ABB RAPID module: Module1.mod

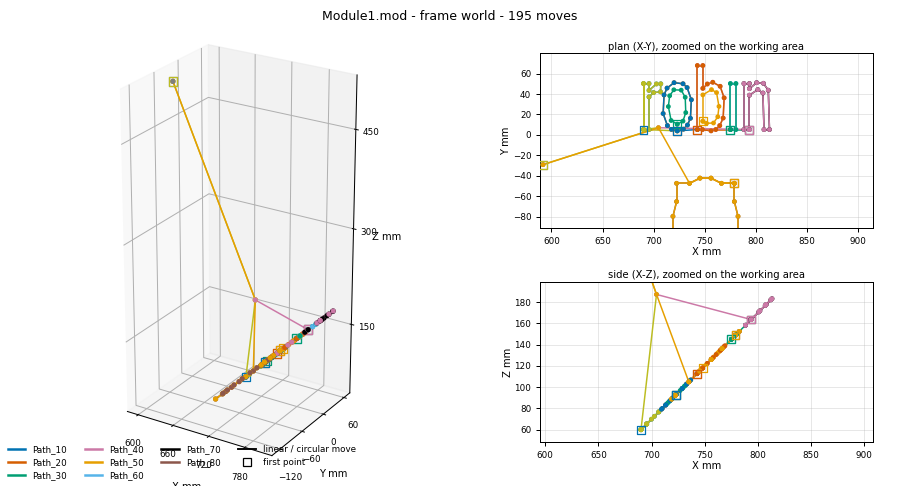
[picture p0: tool path of Module1.mod in frame world, 195 of 195 moves have a stored position in this frame; points joined in program order, loops and branches not executed]
MODULE Module1
        CONST robtarget Target_10:=[[-207.881930308,149.087746467,0.000160807],[0.518535839,0.510701659,-0.288134644,0.622320517],[0,0,1,1],[9E+09,9E+09,9E+09,9E+09,9E+09,9E+09]];
    CONST robtarget Target_20:=[[-247.65501993,195.765129088,0.000181206],[0.450409444,-0.243963603,-0.202089765,-0.83472919],[0,0,0,0],[9E+09,9E+09,9E+09,9E+09,9E+09,9E+09]];
    CONST robtarget Target_30:=[[-247.65501993,188.180039946,0.000181208],[0.450409444,-0.243963603,-0.202089765,-0.83472919],[0,0,0,0],[9E+09,9E+09,9E+09,9E+09,9E+09,9E+09]];
    CONST robtarget Target_40:=[[-240.945133383,188.180039946,0.000181208],[0.450409444,-0.243963603,-0.202089765,-0.83472919],[0,0,0,0],[9E+09,9E+09,9E+09,9E+09,9E+09,9E+09]];
    CONST robtarget Target_50:=[[-247.278196592,177.914642864,0.000181211],[0.450409444,-0.243963603,-0.202089765,-0.83472919],[0,0,0,0],[9E+09,9E+09,9E+09,9E+09,9E+09,9E+09]];
    CONST robtarget Target_60:=[[-247.411908099,171.89154724,0.000181212],[0.450409444,-0.243963603,-0.202089765,-0.83472919],[0,0,0,0],[9E+09,9E+09,9E+09,9E+09,9E+09,9E+09]];
    CONST robtarget Target_70:=[[-239.53508476,172.28052617,0.000181212],[0.450409444,-0.243963603,-0.202089765,-0.83472919],[0,0,0,0],[9E+09,9E+09,9E+09,9E+09,9E+09,9E+09]];
    CONST robtarget Target_80:=[[-238.811255907,181.791619828,0.00018121],[0.450409444,-0.243963603,-0.202089765,-0.83472919],[0,0,0,0],[9E+09,9E+09,9E+09,9E+09,9E+09,9E+09]];
    CONST robtarget Target_90:=[[-234.575603399,188.180039946,0.000181208],[0.450409444,-0.243963603,-0.202089765,-0.83472919],[0,0,0,0],[9E+09,9E+09,9E+09,9E+09,9E+09,9E+09]];
    CONST robtarget Target_100:=[[-202.630708747,188.180039946,0.000181208],[0.450409444,-0.243963603,-0.202089765,-0.83472919],[0,0,0,0],[9E+09,9E+09,9E+09,9E+09,9E+09,9E+09]];
    CONST robtarget Target_110:=[[-202.630708747,195.765129088,0.000181206],[0.450409444,-0.243963603,-0.202089765,-0.83472919],[0,0,0,0],[9E+09,9E+09,9E+09,9E+09,9E+09,9E+09]];
    CONST robtarget Target_120:=[[-201.366527224,149.087657451,0.000181219],[0.450409444,-0.243963603,-0.202089765,-0.83472919],[0,0,0,0],[9E+09,9E+09,9E+09,9E+09,9E+09,9E+09]];
    CONST robtarget Target_130:=[[-203.021765343,140.621098181,0.000181221],[0.450409444,-0.243963603,-0.202089765,-0.83472919],[0,0,0,0],[9E+09,9E+09,9E+09,9E+09,9E+09,9E+09]];
    CONST robtarget Target_140:=[[-207.051498291,134.946923266,0.000181223],[0.450409444,-0.243963603,-0.202089765,-0.83472919],[0,0,0,0],[9E+09,9E+09,9E+09,9E+09,9E+09,9E+09]];
    CONST robtarget Target_150:=[[-213.680713864,130.849034031,0.000181224],[0.450409444,-0.243963603,-0.202089765,-0.83472919],[0,0,0,0],[9E+09,9E+09,9E+09,9E+09,9E+09,9E+09]];
    CONST robtarget Target_160:=[[-231.788173899,129.551975923,0.000181224],[0.450409444,-0.243963603,-0.202089765,-0.83472919],[0,0,0,0],[9E+09,9E+09,9E+09,9E+09,9E+09,9E+09]];
    CONST robtarget Target_170:=[[-243.683087922,135.407213167,0.000181223],[0.450409444,-0.243963603,-0.202089765,-0.83472919],[0,0,0,0],[9E+09,9E+09,9E+09,9E+09,9E+09,9E+09]];
    CONST robtarget Target_180:=[[-247.461911379,141.100681452,0.000181221],[0.450409444,-0.243963603,-0.202089765,-0.83472919],[0,0,0,0],[9E+09,9E+09,9E+09,9E+09,9E+09,9E+09]];
    CONST robtarget Target_190:=[[-248.515109012,153.46115467,0.000181218],[0.450409444,-0.243963603,-0.202089765,-0.83472919],[0,0,0,0],[9E+09,9E+09,9E+09,9E+09,9E+09,9E+09]];
    CONST robtarget Target_200:=[[-243.220985991,163.168323786,0.000181215],[0.450409444,-0.243963603,-0.202089765,-0.83472919],[0,0,0,0],[9E+09,9E+09,9E+09,9E+09,9E+09,9E+09]];
    CONST robtarget Target_210:=[[-236.515653903,167.360178067,0.000181214],[0.450409444,-0.243963603,-0.202089765,-0.83472919],[0,0,0,0],[9E+09,9E+09,9E+09,9E+09,9E+09,9E+09]];
    CONST robtarget Target_220:=[[-218.290970645,168.613376793,0.000181213],[0.450409444,-0.243963603,-0.202089765,-0.83472919],[0,0,0,0],[9E+09,9E+09,9E+09,9E+09,9E+09,9E+09]];
    CONST robtarget Target_230:=[[-206.527619769,162.711873191,0.000181215],[0.450409444,-0.243963603,-0.202089765,-0.83472919],[0,0,0,0],[9E+09,9E+09,9E+09,9E+09,9E+09,9E+09]];
    CONST robtarget Target_240:=[[-202.813142148,157.107360988,0.000181217],[0.450409444,-0.243963603,-0.202089765,-0.83472919],[0,0,0,0],[9E+09,9E+09,9E+09,9E+09,9E+09,9E+09]];
    CONST robtarget Target_250:=[[-201.366527224,149.087657451,0.000181219],[0.450409444,-0.243963603,-0.202089765,-0.83472919],[0,0,0,0],[9E+09,9E+09,9E+09,9E+09,9E+09,9E+09]];
    CONST robtarget Target_450:=[[-207.881924306,149.087657451,0.000181219],[0.450409444,-0.243963603,-0.202089765,-0.83472919],[0,0,0,0],[9E+09,9E+09,9E+09,9E+09,9E+09,9E+09]];
    CONST robtarget Target_460:=[[-210.90124058,141.155060399,0.000181221],[0.450409444,-0.243963603,-0.202089765,-0.83472919],[0,0,0,0],[9E+09,9E+09,9E+09,9E+09,9E+09,9E+09]];
    CONST robtarget Target_470:=[[-219.222672222,137.293167892,0.000181222],[0.450409444,-0.243963603,-0.202089765,-0.83472919],[0,0,0,0],[9E+09,9E+09,9E+09,9E+09,9E+09,9E+09]];
    CONST robtarget Target_480:=[[-234.22183773,138.044318657,0.000181223],[0.450409444,-0.243963603,-0.202089765,-0.83472919],[0,0,0,0],[9E+09,9E+09,9E+09,9E+09,9E+09,9E+09]];
    CONST robtarget Target_490:=[[-241.204901386,143.601825103,0.00018122],[0.450409444,-0.243963603,-0.202089765,-0.83472919],[0,0,0,0],[9E+09,9E+09,9E+09,9E+09,9E+09,9E+09]];
    CONST robtarget Target_500:=[[-241.55017581,153.821736994,0.000181218],[0.450409444,-0.243963603,-0.202089765,-0.83472919],[0,0,0,0],[9E+09,9E+09,9E+09,9E+09,9E+09,9E+09]];
    CONST robtarget Target_510:=[[-235.724815439,159.591250126,0.000181216],[0.450409444,-0.243963603,-0.202089765,-0.83472919],[0,0,0,0],[9E+09,9E+09,9E+09,9E+09,9E+09,9E+09]];
    CONST robtarget Target_520:=[[-225.142864339,161.389116121,0.000181215],[0.450409444,-0.243963603,-0.202089765,-0.83472919],[0,0,0,0],[9E+09,9E+09,9E+09,9E+09,9E+09,9E+09]];
    CONST robtarget Target_530:=[[-211.506651645,157.581568731,0.000181217],[0.450409444,-0.243963603,-0.202089765,-0.83472919],[0,0,0,0],[9E+09,9E+09,9E+09,9E+09,9E+09,9E+09]];
    CONST robtarget Target_540:=[[-207.881924306,149.087657451,0.000181219],[0.450409444,-0.243963603,-0.202089765,-0.83472919],[0,0,0,0],[9E+09,9E+09,9E+09,9E+09,9E+09,9E+09]];
    CONST robtarget Target_550:=[[-202.630708747,121.227041567,0.000181228],[0.450409444,-0.243963603,-0.202089765,-0.83472919],[0,0,0,0],[9E+09,9E+09,9E+09,9E+09,9E+09,9E+09]];
    CONST robtarget Target_560:=[[-202.630708747,114.128176089,0.000181229],[0.450409444,-0.243963603,-0.202089765,-0.83472919],[0,0,0,0],[9E+09,9E+09,9E+09,9E+09,9E+09,9E+09]];
    CONST robtarget Target_570:=[[-201.366527224,102.264318715,0.000181232],[0.450409444,-0.243963603,-0.202089765,-0.83472919],[0,0,0,0],[9E+09,9E+09,9E+09,9E+09,9E+09,9E+09]];
    CONST robtarget Target_580:=[[-202.647957508,95.740722444,0.000181234],[0.450409444,-0.243963603,-0.202089765,-0.83472919],[0,0,0,0],[9E+09,9E+09,9E+09,9E+09,9E+09,9E+09]];
    CONST robtarget Target_590:=[[-206.492248362,90.253373046,0.000181236],[0.450409444,-0.243963603,-0.202089765,-0.83472919],[0,0,0,0],[9E+09,9E+09,9E+09,9E+09,9E+09,9E+09]];
    CONST robtarget Target_600:=[[-213.89225132,85.531430921,0.000181237],[0.450409444,-0.243963603,-0.202089765,-0.83472919],[0,0,0,0],[9E+09,9E+09,9E+09,9E+09,9E+09,9E+09]];
    CONST robtarget Target_610:=[[-233.637220258,84.167137,0.000181237],[0.450409444,-0.243963603,-0.202089765,-0.83472919],[0,0,0,0],[9E+09,9E+09,9E+09,9E+09,9E+09,9E+09]];
    CONST robtarget Target_620:=[[-244.963719116,89.701429516,0.000181236],[0.450409444,-0.243963603,-0.202089765,-0.83472919],[0,0,0,0],[9E+09,9E+09,9E+09,9E+09,9E+09,9E+09]];
    CONST robtarget Target_630:=[[-248.919201454,99.881822767,0.000181233],[0.450409444,-0.243963603,-0.202089765,-0.83472919],[0,0,0,0],[9E+09,9E+09,9E+09,9E+09,9E+09,9E+09]];
    CONST robtarget Target_640:=[[-247.217418634,107.442600725,0.000181231],[0.450409444,-0.243963603,-0.202089765,-0.83472919],[0,0,0,0],[9E+09,9E+09,9E+09,9E+09,9E+09,9E+09]];
    CONST robtarget Target_650:=[[-242.9386504,113.641952426,0.000181229],[0.450409444,-0.243963603,-0.202089765,-0.83472919],[0,0,0,0],[9E+09,9E+09,9E+09,9E+09,9E+09,9E+09]];
    CONST robtarget Target_660:=[[-265.304938893,113.641952426,0.000181229],[0.450409444,-0.243963603,-0.202089765,-0.83472919],[0,0,0,0],[9E+09,9E+09,9E+09,9E+09,9E+09,9E+09]];
    CONST robtarget Target_670:=[[-265.304938893,121.227041567,0.000181228],[0.450409444,-0.243963603,-0.202089765,-0.83472919],[0,0,0,0],[9E+09,9E+09,9E+09,9E+09,9E+09,9E+09]];
    CONST robtarget Target_680:=[[-202.630708747,121.227041567,0.000181228],[0.450409444,-0.243963603,-0.202089765,-0.83472919],[0,0,0,0],[9E+09,9E+09,9E+09,9E+09,9E+09,9E+09]];
    CONST robtarget Target_760:=[[-210.750643917,113.641952426,0.000181229],[0.450409444,-0.243963603,-0.202089765,-0.83472919],[0,0,0,0],[9E+09,9E+09,9E+09,9E+09,9E+09,9E+09]];
    CONST robtarget Target_770:=[[-236.569120417,113.641952426,0.000181229],[0.450409444,-0.243963603,-0.202089765,-0.83472919],[0,0,0,0],[9E+09,9E+09,9E+09,9E+09,9E+09,9E+09]];
    CONST robtarget Target_780:=[[-241.723091243,101.68085032,0.000181232],[0.450409444,-0.243963603,-0.202089765,-0.83472919],[0,0,0,0],[9E+09,9E+09,9E+09,9E+09,9E+09,9E+09]];
    CONST robtarget Target_790:=[[-238.824332003,94.685562215,0.000181234],[0.450409444,-0.243963603,-0.202089765,-0.83472919],[0,0,0,0],[9E+09,9E+09,9E+09,9E+09,9E+09,9E+09]];
    CONST robtarget Target_800:=[[-225.288731438,91.3242863,0.000181235],[0.450409444,-0.243963603,-0.202089765,-0.83472919],[0,0,0,0],[9E+09,9E+09,9E+09,9E+09,9E+09,9E+09]];
    CONST robtarget Target_810:=[[-215.163302593,92.950711075,0.000181235],[0.450409444,-0.243963603,-0.202089765,-0.83472919],[0,0,0,0],[9E+09,9E+09,9E+09,9E+09,9E+09,9E+09]];
    CONST robtarget Target_820:=[[-209.047609429,98.913303675,0.000181233],[0.450409444,-0.243963603,-0.202089765,-0.83472919],[0,0,0,0],[9E+09,9E+09,9E+09,9E+09,9E+09,9E+09]];
    CONST robtarget Target_830:=[[-208.7571269,108.560915149,0.00018123],[0.450409444,-0.243963603,-0.202089765,-0.83472919],[0,0,0,0],[9E+09,9E+09,9E+09,9E+09,9E+09,9E+09]];
    CONST robtarget Target_840:=[[-210.750643917,113.641952426,0.000181229],[0.450409444,-0.243963603,-0.202089765,-0.83472919],[0,0,0,0],[9E+09,9E+09,9E+09,9E+09,9E+09,9E+09]];
    CONST robtarget Target_850:=[[-202.630708747,75.47339489,0.00018124],[0.450409444,-0.243963603,-0.202089765,-0.83472919],[0,0,0,0],[9E+09,9E+09,9E+09,9E+09,9E+09,9E+09]];
    CONST robtarget Target_860:=[[-247.65501993,75.47339489,0.00018124],[0.450409444,-0.243963603,-0.202089765,-0.83472919],[0,0,0,0],[9E+09,9E+09,9E+09,9E+09,9E+09,9E+09]];
    CONST robtarget Target_870:=[[-247.65501993,67.888305748,0.000181242],[0.450409444,-0.243963603,-0.202089765,-0.83472919],[0,0,0,0],[9E+09,9E+09,9E+09,9E+09,9E+09,9E+09]];
    CONST robtarget Target_880:=[[-202.630708747,67.888305748,0.000181242],[0.450409444,-0.243963603,-0.202089765,-0.83472919],[0,0,0,0],[9E+09,9E+09,9E+09,9E+09,9E+09,9E+09]];
    CONST robtarget Target_890:=[[-202.630708747,75.47339489,0.00018124],[0.450409444,-0.243963603,-0.202089765,-0.83472919],[0,0,0,0],[9E+09,9E+09,9E+09,9E+09,9E+09,9E+09]];
    CONST robtarget Target_900:=[[-202.630708747,49.168694728,0.000181247],[0.450409444,-0.243963603,-0.202089765,-0.83472919],[0,0,0,0],[9E+09,9E+09,9E+09,9E+09,9E+09,9E+09]];
    CONST robtarget Target_910:=[[-202.630708747,56.753783869,0.000181245],[0.450409444,-0.243963603,-0.202089765,-0.83472919],[0,0,0,0],[9E+09,9E+09,9E+09,9E+09,9E+09,9E+09]];
    CONST robtarget Target_920:=[[-247.65501993,56.753783869,0.000181245],[0.450409444,-0.243963603,-0.202089765,-0.83472919],[0,0,0,0],[9E+09,9E+09,9E+09,9E+09,9E+09,9E+09]];
    CONST robtarget Target_930:=[[-247.65501993,49.168694728,0.000181247],[0.450409444,-0.243963603,-0.202089765,-0.83472919],[0,0,0,0],[9E+09,9E+09,9E+09,9E+09,9E+09,9E+09]];
    CONST robtarget Target_940:=[[-242.646916203,49.168694728,0.000181247],[0.450409444,-0.243963603,-0.202089765,-0.83472919],[0,0,0,0],[9E+09,9E+09,9E+09,9E+09,9E+09,9E+09]];
    CONST robtarget Target_950:=[[-248.518066932,39.09778711,0.00018125],[0.450409444,-0.243963603,-0.202089765,-0.83472919],[0,0,0,0],[9E+09,9E+09,9E+09,9E+09,9E+09,9E+09]];
    CONST robtarget Target_960:=[[-247.89555783,29.780399186,0.000181253],[0.450409444,-0.243963603,-0.202089765,-0.83472919],[0,0,0,0],[9E+09,9E+09,9E+09,9E+09,9E+09,9E+09]];
    CONST robtarget Target_970:=[[-241.106205462,23.03357744,0.000181255],[0.450409444,-0.243963603,-0.202089765,-0.83472919],[0,0,0,0],[9E+09,9E+09,9E+09,9E+09,9E+09,9E+09]];
    CONST robtarget Target_980:=[[-202.630708747,21.405323577,0.000181255],[0.450409444,-0.243963603,-0.202089765,-0.83472919],[0,0,0,0],[9E+09,9E+09,9E+09,9E+09,9E+09,9E+09]];
    CONST robtarget Target_990:=[[-202.630708747,28.990412718,0.000181253],[0.450409444,-0.243963603,-0.202089765,-0.83472919],[0,0,0,0],[9E+09,9E+09,9E+09,9E+09,9E+09,9E+09]];
    CONST robtarget Target_1000:=[[-238.368147969,30.449083707,0.000181253],[0.450409444,-0.243963603,-0.202089765,-0.83472919],[0,0,0,0],[9E+09,9E+09,9E+09,9E+09,9E+09,9E+09]];
    CONST robtarget Target_1010:=[[-241.723091243,37.499326818,0.000181251],[0.450409444,-0.243963603,-0.202089765,-0.83472919],[0,0,0,0],[9E+09,9E+09,9E+09,9E+09,9E+09,9E+09]];
    CONST robtarget Target_1020:=[[-236.277386219,49.168694728,0.000181247],[0.450409444,-0.243963603,-0.202089765,-0.83472919],[0,0,0,0],[9E+09,9E+09,9E+09,9E+09,9E+09,9E+09]];
    CONST robtarget Target_1030:=[[-202.630708747,49.168694728,0.000181247],[0.450409444,-0.243963603,-0.202089765,-0.83472919],[0,0,0,0],[9E+09,9E+09,9E+09,9E+09,9E+09,9E+09]];
    CONST robtarget Target_1240:=[[-149.999876139,69.999739674,0.000181241],[0.450409444,-0.243963603,-0.202089765,-0.83472919],[0,0,0,0],[9E+09,9E+09,9E+09,9E+09,9E+09,9E+09]];
    CONST robtarget Target_1250:=[[-149.999876139,87.894319411,0.000181236],[0.450409444,-0.243963603,-0.202089765,-0.83472919],[0,0,0,0],[9E+09,9E+09,9E+09,9E+09,9E+09,9E+09]];
    CONST robtarget Target_1260:=[[-155.055991083,102.344929998,0.000181232],[0.450409444,-0.243963603,-0.202089765,-0.83472919],[0,0,0,0],[9E+09,9E+09,9E+09,9E+09,9E+09,9E+09]];
    CONST robtarget Target_1270:=[[-155.055991083,117.65454935,0.000181228],[0.450409444,-0.243963603,-0.202089765,-0.83472919],[0,0,0,0],[9E+09,9E+09,9E+09,9E+09,9E+09,9E+09]];
    CONST robtarget Target_1280:=[[-149.999876139,132.105159938,0.000181224],[0.450409444,-0.243963603,-0.202089765,-0.83472919],[0,0,0,0],[9E+09,9E+09,9E+09,9E+09,9E+09,9E+09]];
    CONST robtarget Target_1290:=[[-149.999876139,149.999739674,0.000181219],[0.450409444,-0.243963603,-0.202089765,-0.83472919],[0,0,0,0],[9E+09,9E+09,9E+09,9E+09,9E+09,9E+09]];
    CONST robtarget Target_1300:=[[-132.105296402,149.999739674,0.000181219],[0.450409444,-0.243963603,-0.202089765,-0.83472919],[0,0,0,0],[9E+09,9E+09,9E+09,9E+09,9E+09,9E+09]];
    CONST robtarget Target_1310:=[[-117.654685815,155.055854619,0.000181218],[0.450409444,-0.243963603,-0.202089765,-0.83472919],[0,0,0,0],[9E+09,9E+09,9E+09,9E+09,9E+09,9E+09]];
    CONST robtarget Target_1320:=[[-102.345066463,155.055854619,0.000181218],[0.450409444,-0.243963603,-0.202089765,-0.83472919],[0,0,0,0],[9E+09,9E+09,9E+09,9E+09,9E+09,9E+09]];
    CONST robtarget Target_1330:=[[-87.894455875,149.999739674,0.000181219],[0.450409444,-0.243963603,-0.202089765,-0.83472919],[0,0,0,0],[9E+09,9E+09,9E+09,9E+09,9E+09,9E+09]];
    CONST robtarget Target_1340:=[[-69.999876139,149.999739674,0.000181219],[0.450409444,-0.243963603,-0.202089765,-0.83472919],[0,0,0,0],[9E+09,9E+09,9E+09,9E+09,9E+09,9E+09]];
    CONST robtarget Target_1350:=[[-69.999876139,132.105159938,0.000181224],[0.450409444,-0.243963603,-0.202089765,-0.83472919],[0,0,0,0],[9E+09,9E+09,9E+09,9E+09,9E+09,9E+09]];
    CONST robtarget Target_1360:=[[-64.943761195,117.65454935,0.000181228],[0.450409444,-0.243963603,-0.202089765,-0.83472919],[0,0,0,0],[9E+09,9E+09,9E+09,9E+09,9E+09,9E+09]];
    CONST robtarget Target_1370:=[[-64.943761195,102.344929998,0.000181232],[0.450409444,-0.243963603,-0.202089765,-0.83472919],[0,0,0,0],[9E+09,9E+09,9E+09,9E+09,9E+09,9E+09]];
    CONST robtarget Target_1380:=[[-69.999876139,87.894319411,0.000181236],[0.450409444,-0.243963603,-0.202089765,-0.83472919],[0,0,0,0],[9E+09,9E+09,9E+09,9E+09,9E+09,9E+09]];
    CONST robtarget Target_1390:=[[-69.999876139,69.999739674,0.000181241],[0.450409444,-0.243963603,-0.202089765,-0.83472919],[0,0,0,0],[9E+09,9E+09,9E+09,9E+09,9E+09,9E+09]];
    CONST robtarget Target_1400:=[[-87.894455875,69.999739674,0.000181241],[0.450409444,-0.243963603,-0.202089765,-0.83472919],[0,0,0,0],[9E+09,9E+09,9E+09,9E+09,9E+09,9E+09]];
    CONST robtarget Target_1410:=[[-102.345066463,64.943624731,0.000181243],[0.450409444,-0.243963603,-0.202089765,-0.83472919],[0,0,0,0],[9E+09,9E+09,9E+09,9E+09,9E+09,9E+09]];
    CONST robtarget Target_1420:=[[-117.654685815,64.943624731,0.000181243],[0.450409444,-0.243963603,-0.202089765,-0.83472919],[0,0,0,0],[9E+09,9E+09,9E+09,9E+09,9E+09,9E+09]];
    CONST robtarget Target_1430:=[[-132.105296402,69.999739674,0.000181241],[0.450409444,-0.243963603,-0.202089765,-0.83472919],[0,0,0,0],[9E+09,9E+09,9E+09,9E+09,9E+09,9E+09]];
    CONST robtarget Target_1440:=[[-149.999876139,69.999739674,0.000181241],[0.450409444,-0.243963603,-0.202089765,-0.83472919],[0,0,0,0],[9E+09,9E+09,9E+09,9E+09,9E+09,9E+09]];
    CONST robtarget homeRobot:=[[591.673986457,-29.08667,508.708742654],[0.5,0,0.866025404,0],[0,-1,0,0],[9E+09,9E+09,9E+09,9E+09,9E+09,9E+09]];
    CONST robtarget home_tablero:=[[-204.411694147,95.431074715,-79.679660549],[0.450409444,-0.243963603,-0.202089765,-0.83472919],[-1,-1,1,0],[9E+09,9E+09,9E+09,9E+09,9E+09,9E+09]];
    PERS tooldata robin:=[TRUE,[[105.2184,-29.08667,159.3389],[1,0,0,0]],[0.1,[0,0,1],[1,0,0,0],1,1,1]];
    TASK PERS wobjdata tablero:=[FALSE,TRUE,"",[[828.53,-197.368,198.466],[0.27059805,-0.653281482,0.653281482,-0.27059805]],[[0,0,0],[1,0,0,0]]];
!***********************************************************
    !
    ! Módulo:  Module1
    !
    ! Descripción:
    !   <Introduzca la descripción aquí>
    !
    ! Autor: robin
    !
    ! Versión: 1.0
    !
    !***********************************************************


    !***********************************************************
    !
    ! Procedimiento Main
    !
    !   Este es el punto de entrada de su programa
    !
    !***********************************************************
    PROC main()
        !Añada aquí su código
        letra_r;
        letra_o;
        letra_b;
        letra_i;
        letra_n;
        decoracion;
    ENDPROC
    PROC Path_10()
         MoveL Target_110,v100,z100,robin\WObj:=tablero;
        MoveL Target_20,v100,z100,robin\WObj:=tablero;
         MoveL Target_30,v100,z100,robin\WObj:=tablero;
          MoveL Target_40,v100,z100,robin\WObj:=tablero;
           MoveL Target_50,v100,z100,robin\WObj:=tablero;
            MoveL Target_60,v100,z100,robin\WObj:=tablero;
             MoveL Target_70,v100,z100,robin\WObj:=tablero;
              MoveL Target_80,v100,z100,robin\WObj:=tablero;
               MoveL Target_90,v100,z100,robin\WObj:=tablero;
                MoveL Target_100,v100,z100,robin\WObj:=tablero;

        MoveL Target_110,v100,z100,robin\WObj:=tablero;
    ENDPROC
    PROC Path_20()
        MoveL Target_120,v100,z100,robin\WObj:=tablero;
        MoveL Target_130,v100,z100,robin\WObj:=tablero;
        MoveL Target_140,v100,z100,robin\WObj:=tablero;
        MoveL Target_150,v100,z100,robin\WObj:=tablero;
        MoveL Target_160,v100,z100,robin\WObj:=tablero;
        MoveL Target_170,v100,z100,robin\WObj:=tablero;
        MoveL Target_180,v100,z100,robin\WObj:=tablero;
        MoveL Target_190,v100,z100,robin\WObj:=tablero;
        MoveL Target_200,v100,z100,robin\WObj:=tablero;
        MoveL Target_210,v100,z100,robin\WObj:=tablero;
        MoveL Target_220,v100,z100,robin\WObj:=tablero;
        MoveL Target_230,v100,z100,robin\WObj:=tablero;
        MoveL Target_240,v100,z100,robin\WObj:=tablero;
        MoveL Target_250,v100,z100,robin\WObj:=tablero;
    ENDPROC
    PROC Path_30()
        MoveL Target_450,v100,z100,robin\WObj:=tablero;
        MoveL Target_460,v100,z100,robin\WObj:=tablero;
        MoveL Target_470,v100,z100,robin\WObj:=tablero;
        MoveL Target_480,v100,z100,robin\WObj:=tablero;
        MoveL Target_490,v100,z100,robin\WObj:=tablero;
        MoveL Target_500,v100,z100,robin\WObj:=tablero;
        MoveL Target_510,v100,z100,robin\WObj:=tablero;
        MoveL Target_520,v100,z100,robin\WObj:=tablero;
        MoveL Target_530,v100,z100,robin\WObj:=tablero;
        MoveL Target_540,v100,z100,robin\WObj:=tablero;
    ENDPROC
    PROC Path_40()
        MoveL Target_550,v100,z100,robin\WObj:=tablero;
        MoveL Target_560,v100,z100,robin\WObj:=tablero;
        MoveL Target_570,v100,z100,robin\WObj:=tablero;
        MoveL Target_580,v100,z100,robin\WObj:=tablero;
        MoveL Target_590,v100,z100,robin\WObj:=tablero;
        MoveL Target_600,v100,z100,robin\WObj:=tablero;
        MoveL Target_610,v100,z100,robin\WObj:=tablero;
        MoveL Target_620,v100,z100,robin\WObj:=tablero;
        MoveL Target_630,v100,z100,robin\WObj:=tablero;
        MoveL Target_640,v100,z100,robin\WObj:=tablero;
        MoveL Target_650,v100,z100,robin\WObj:=tablero;
        MoveL Target_660,v100,z100,robin\WObj:=tablero;
        MoveL Target_670,v100,z100,robin\WObj:=tablero;
        MoveL Target_680,v100,z100,robin\WObj:=tablero;
    ENDPROC
    PROC Path_50()
        MoveL Target_760,v100,z100,robin\WObj:=tablero;
        MoveL Target_770,v100,z100,robin\WObj:=tablero;
        MoveL Target_780,v100,z100,robin\WObj:=tablero;
        MoveL Target_790,v100,z100,robin\WObj:=tablero;
        MoveL Target_800,v100,z100,robin\WObj:=tablero;
        MoveL Target_810,v100,z100,robin\WObj:=tablero;
        MoveL Target_820,v100,z100,robin\WObj:=tablero;
        MoveL Target_830,v100,z100,robin\WObj:=tablero;
        MoveL Target_840,v100,z100,robin\WObj:=tablero;
    ENDPROC
    PROC Path_60()
        MoveL Target_850,v100,z100,robin\WObj:=tablero;
        MoveL Target_860,v100,z100,robin\WObj:=tablero;
        MoveL Target_870,v100,z100,robin\WObj:=tablero;
        MoveL Target_880,v100,z100,robin\WObj:=tablero;
        MoveL Target_890,v100,z100,robin\WObj:=tablero;
    ENDPROC
    PROC Path_70()
        MoveL Target_900,v100,z100,robin\WObj:=tablero;
        MoveL Target_910,v100,z100,robin\WObj:=tablero;
        MoveL Target_920,v100,z100,robin\WObj:=tablero;
        MoveL Target_930,v100,z100,robin\WObj:=tablero;
        MoveL Target_940,v100,z100,robin\WObj:=tablero;
        MoveL Target_950,v100,z100,robin\WObj:=tablero;
        MoveL Target_960,v100,z100,robin\WObj:=tablero;
        MoveL Target_970,v100,z100,robin\WObj:=tablero;
        MoveL Target_980,v100,z100,robin\WObj:=tablero;
        MoveL Target_990,v100,z100,robin\WObj:=tablero;
        MoveL Target_1000,v100,z100,robin\WObj:=tablero;
        MoveL Target_1010,v100,z100,robin\WObj:=tablero;
        MoveL Target_1020,v100,z100,robin\WObj:=tablero;
        MoveL Target_1030,v100,z100,robin\WObj:=tablero;
    ENDPROC
    PROC Path_80()
        MoveL Target_1240,v100,z100,robin\WObj:=tablero;
        MoveL Target_1250,v100,z100,robin\WObj:=tablero;
        MoveL Target_1260,v100,z100,robin\WObj:=tablero;
        MoveL Target_1270,v100,z100,robin\WObj:=tablero;
        MoveL Target_1280,v100,z100,robin\WObj:=tablero;
        MoveL Target_1290,v100,z100,robin\WObj:=tablero;
        MoveL Target_1300,v100,z100,robin\WObj:=tablero;
        MoveL Target_1310,v100,z100,robin\WObj:=tablero;
        MoveL Target_1320,v100,z100,robin\WObj:=tablero;
        MoveL Target_1330,v100,z100,robin\WObj:=tablero;
        MoveL Target_1340,v100,z100,robin\WObj:=tablero;
        MoveL Target_1350,v100,z100,robin\WObj:=tablero;
        MoveL Target_1360,v100,z100,robin\WObj:=tablero;
        MoveL Target_1370,v100,z100,robin\WObj:=tablero;
        MoveL Target_1380,v100,z100,robin\WObj:=tablero;
        MoveL Target_1390,v100,z100,robin\WObj:=tablero;
        MoveL Target_1400,v100,z100,robin\WObj:=tablero;
        MoveL Target_1410,v100,z100,robin\WObj:=tablero;
        MoveL Target_1420,v100,z100,robin\WObj:=tablero;
        MoveL Target_1430,v100,z100,robin\WObj:=tablero;
        MoveL Target_1440,v100,z100,robin\WObj:=tablero;
    ENDPROC
    PROC Path_90()
        MoveL homeRobot,v100,z100,robin\WObj:=wobj0;
        Path_80;
    ENDPROC
    PROC letra_r()
        MoveL homeRobot,v100,z100,robin\WObj:=wobj0;
        MoveL home_tablero,v100,z1,robin\WObj:=tablero;
        MoveL Target_110,v100,z100,robin\WObj:=tablero;
        MoveL Target_20,v100,z100,robin\WObj:=tablero;
         MoveL Target_110,v100,z100,robin\WObj:=tablero;
        MoveL Target_20,v100,z100,robin\WObj:=tablero;
        MoveL Target_30,v100,z100,robin\WObj:=tablero;
        MoveL Target_40,v100,z100,robin\WObj:=tablero;
        MoveL Target_50,v100,z100,robin\WObj:=tablero;
        MoveL Target_60,v100,z100,robin\WObj:=tablero;
        MoveL Target_70,v100,z100,robin\WObj:=tablero;
        MoveL Target_80,v100,z100,robin\WObj:=tablero;
        MoveL Target_90,v100,z100,robin\WObj:=tablero;
        MoveL Target_100,v100,z100,robin\WObj:=tablero;
        MoveL Target_110,v100,z100,robin\WObj:=tablero;
        MoveL Target_120,v100,z100,robin\WObj:=tablero;
    ENDPROC
    PROC letra_o()
        MoveL Target_120,v100,z100,robin\WObj:=tablero;
        MoveL Target_130,v100,z100,robin\WObj:=tablero;
        MoveL Target_140,v100,z100,robin\WObj:=tablero;
        MoveL Target_150,v100,z100,robin\WObj:=tablero;
        MoveL Target_160,v100,z100,robin\WObj:=tablero;
        MoveL Target_170,v100,z100,robin\WObj:=tablero;
        MoveL Target_180,v100,z100,robin\WObj:=tablero;
        MoveL Target_190,v100,z100,robin\WObj:=tablero;
        MoveL Target_200,v100,z100,robin\WObj:=tablero;
        MoveL Target_210,v100,z100,robin\WObj:=tablero;
        MoveL Target_220,v100,z100,robin\WObj:=tablero;
        MoveL Target_230,v100,z100,robin\WObj:=tablero;
        MoveL Target_240,v100,z100,robin\WObj:=tablero;
        MoveL Target_250,v100,z100,robin\WObj:=tablero;
        MoveL Target_550,v1000,z100,robin\WObj:=tablero;
    ENDPROC
    PROC letra_b()
        MoveL Target_550,v100,z100,robin\WObj:=tablero;
        MoveL Target_560,v100,z100,robin\WObj:=tablero;
        MoveL Target_570,v100,z100,robin\WObj:=tablero;
        MoveL Target_580,v100,z100,robin\WObj:=tablero;
        MoveL Target_590,v100,z100,robin\WObj:=tablero;
        MoveL Target_600,v100,z100,robin\WObj:=tablero;
        MoveL Target_610,v100,z100,robin\WObj:=tablero;
        MoveL Target_620,v100,z100,robin\WObj:=tablero;
        MoveL Target_630,v100,z100,robin\WObj:=tablero;
        MoveL Target_640,v100,z100,robin\WObj:=tablero;
        MoveL Target_650,v100,z100,robin\WObj:=tablero;
        MoveL Target_660,v100,z100,robin\WObj:=tablero;
        MoveL Target_670,v100,z100,robin\WObj:=tablero;
        MoveL Target_680,v100,z100,robin\WObj:=tablero;
        MoveL Target_850,v100,z100,robin\WObj:=tablero;
    ENDPROC
    PROC letra_i()
        MoveL Target_850,v100,z100,robin\WObj:=tablero;
        MoveL Target_860,v100,z100,robin\WObj:=tablero;
        MoveL Target_870,v100,z100,robin\WObj:=tablero;
        MoveL Target_880,v100,z100,robin\WObj:=tablero;
        MoveL Target_890,v100,z100,robin\WObj:=tablero;
        MoveL Target_850,v1000,z100,robin\WObj:=tablero;
        MoveL Target_900,v100,z100,robin\WObj:=tablero;
    ENDPROC
    PROC letra_n()
        MoveL Target_900,v100,z100,robin\WObj:=tablero;
        MoveL Target_910,v100,z100,robin\WObj:=tablero;
        MoveL Target_920,v100,z100,robin\WObj:=tablero;
        MoveL Target_930,v100,z100,robin\WObj:=tablero;
        MoveL Target_940,v100,z100,robin\WObj:=tablero;
        MoveL Target_950,v100,z100,robin\WObj:=tablero;
        MoveL Target_960,v100,z100,robin\WObj:=tablero;
        MoveL Target_970,v100,z100,robin\WObj:=tablero;
        MoveL Target_980,v100,z100,robin\WObj:=tablero;
        MoveL Target_990,v100,z100,robin\WObj:=tablero;
        MoveL Target_1000,v100,z100,robin\WObj:=tablero;
        MoveL Target_1010,v100,z100,robin\WObj:=tablero;
        MoveL Target_1020,v100,z100,robin\WObj:=tablero;
        MoveL Target_1030,v100,z100,robin\WObj:=tablero;
        MoveL home_tablero,v100,z100,robin\WObj:=tablero;
    ENDPROC
    PROC decoracion()
        MoveL Target_1240,v100,z100,robin\WObj:=tablero;
        MoveL Target_1250,v100,z100,robin\WObj:=tablero;
        MoveL Target_1260,v100,z100,robin\WObj:=tablero;
        MoveL Target_1270,v100,z100,robin\WObj:=tablero;
        MoveL Target_1280,v100,z100,robin\WObj:=tablero;
        MoveL Target_1290,v100,z100,robin\WObj:=tablero;
        MoveL Target_1300,v100,z100,robin\WObj:=tablero;
        MoveL Target_1310,v100,z100,robin\WObj:=tablero;
        MoveL Target_1320,v100,z100,robin\WObj:=tablero;
        MoveL Target_1330,v100,z100,robin\WObj:=tablero;
        MoveL Target_1340,v100,z100,robin\WObj:=tablero;
        MoveL Target_1350,v100,z100,robin\WObj:=tablero;
        MoveL Target_1360,v100,z100,robin\WObj:=tablero;
        MoveL Target_1370,v100,z100,robin\WObj:=tablero;
        MoveL Target_1380,v100,z100,robin\WObj:=tablero;
        MoveL Target_1390,v100,z100,robin\WObj:=tablero;
        MoveL Target_1400,v100,z100,robin\WObj:=tablero;
        MoveL Target_1410,v100,z100,robin\WObj:=tablero;
        MoveL Target_1420,v100,z100,robin\WObj:=tablero;
        MoveL Target_1430,v100,z100,robin\WObj:=tablero;
        MoveL Target_1440,v100,z100,robin\WObj:=tablero;
         MoveL Target_1240,v100,z100,robin\WObj:=tablero;
        MoveL Target_1250,v100,z100,robin\WObj:=tablero;
        MoveL Target_1260,v100,z100,robin\WObj:=tablero;
        MoveL Target_1270,v100,z100,robin\WObj:=tablero;
        MoveL Target_1280,v100,z100,robin\WObj:=tablero;
        MoveL home_tablero,v100,z100,robin\WObj:=tablero;
        MoveL homeRobot,v100,z100,robin\WObj:=wobj0;
    ENDPROC
ENDMODULE
